Fanuc KAREL source: IO0092.KL

-- PROVISIONAL review KL for V1013-1; original PC SHA256 c053603bc9c13fd2113c0ec3fa11f7cea26cb07c266a9dcb957f6e374e9aa121
-- Incomplete behavior may be omitted. Consult companion uncertainty JSON. Do not deploy.
PROGRAM IO0092
%NOLOCKGROUP
-- UNRESOLVED_LOCAL_POOL 5 cells at code offset 13; source declarations unknown
-- DIRECT_LOCAL_WORD_ACCESS alone does not prove INTEGER, REAL, or BOOLEAN
BEGIN
  -- UNRESOLVED_PC offsets 0-18; opcodes 2B,2C,7B
  -- UNRESOLVED_PC offsets 23-30; opcodes 9D,23
  -- UNRESOLVED_PC offsets 35-49; opcodes 2E,22,9D,33,35
  -- UNRESOLVED_PC offsets 54-61; opcodes 9D,23
  -- UNRESOLVED_PC offsets 66-77; opcodes 2E,23
  -- UNRESOLVED_PC offsets 82-105; opcodes 22,21,33,34,19,64,23
  -- UNRESOLVED_PC offsets 110-114; opcodes 7F
  -- UNRESOLVED_PC offsets 119-123; opcodes 27,AA
  -- UNRESOLVED_PC offsets 128-132; opcodes 7F
END IO0092
